{attribute addProperty BoxType "EK1100-0000-0018"}
{attribute addProperty Id "Beckhoff_EL73xxEK1122Beckhoff_EL73xxEK1122_FBF14708162A_0001_EL7332_0000_0016EL7332_BC9603EB19424.25A_0002_EL7332_0000_0017EL7332_BC9603EB19424.25A_0003_EL7332_0000_0018EL7332_BC9603EB19424.25A_0004_EL7332_0000_0019EL7332_BC9603EB19424.25A_0005_EL7332_0000_0020EL7332_BC9603EB19424.25A_0006_EL7332_0000_0021EL7332_BC9603EB19424.25A_0007_EL7332_0000_0022EL7332_BC9603EB19424.25A_0008_EL7332_0000_0023EL7332_20B9391519424.25A_0009_EL7332_0000_0024EL7332_20B9391519424.25A_0010_EL7342_0000_0016EL7342_E03DC37137046.25A_0011_EL7342_0000_0017EL7342_E03DC37137046.25A_0012_EL7342_0000_0018EL7342_E03DC37137046.25A_0013_EL7342_0000_0019EL7342_E03DC37137046.25A_0014_EL7342_0000_0020EL7342_E2585B8337046.25A_0015_EL7342_0000_0021EL7342_E2585B8337046.25A_0016_EL7342_0000_0022EL7342_E2585B8337046.25A_0017_EL7342_0000_0023EL7342_D8FCBEED37046.25A_0018_EL7342_0035_0019EL7342_E03DC37137046.25A_0019_EL7342_0035_0020EL7342_E03DC37137046.25"}
{attribute addProperty CRC "2633030660"}
{attribute addProperty SizeInBites "5462"}
{attribute addProperty SizeInBytes "682.75"}
TYPE Beckhoff_EL73xx_9CF0DC04 EXTENDS EK1100_179A0949 :
STRUCT
	{attribute addProperty Name "Beckhoff_EL73xxEK1122"}
	Beckhoff_EL73xxEK1122 : Beckhoff_EL73xxEK1122_FBF14708;
	{attribute addProperty Name "A_0001_EL7332_0000_0016"}
	A_0001_EL7332_0000_0016 : EL7332_BC9603EB;
	{attribute addProperty Name "A_0002_EL7332_0000_0017"}
	A_0002_EL7332_0000_0017 : EL7332_BC9603EB;
	{attribute addProperty Name "A_0003_EL7332_0000_0018"}
	A_0003_EL7332_0000_0018 : EL7332_BC9603EB;
	{attribute addProperty Name "A_0004_EL7332_0000_0019"}
	A_0004_EL7332_0000_0019 : EL7332_BC9603EB;
	{attribute addProperty Name "A_0005_EL7332_0000_0020"}
	A_0005_EL7332_0000_0020 : EL7332_BC9603EB;
	{attribute addProperty Name "A_0006_EL7332_0000_0021"}
	A_0006_EL7332_0000_0021 : EL7332_BC9603EB;
	{attribute addProperty Name "A_0007_EL7332_0000_0022"}
	A_0007_EL7332_0000_0022 : EL7332_BC9603EB;
	{attribute addProperty Name "A_0008_EL7332_0000_0023"}
	A_0008_EL7332_0000_0023 : EL7332_20B93915;
	{attribute addProperty Name "A_0009_EL7332_0000_0024"}
	A_0009_EL7332_0000_0024 : EL7332_20B93915;
	{attribute addProperty Name "A_0010_EL7342_0000_0016"}
	A_0010_EL7342_0000_0016 : EL7342_E03DC371;
	{attribute addProperty Name "A_0011_EL7342_0000_0017"}
	A_0011_EL7342_0000_0017 : EL7342_E03DC371;
	{attribute addProperty Name "A_0012_EL7342_0000_0018"}
	A_0012_EL7342_0000_0018 : EL7342_E03DC371;
	{attribute addProperty Name "A_0013_EL7342_0000_0019"}
	A_0013_EL7342_0000_0019 : EL7342_E03DC371;
	{attribute addProperty Name "A_0014_EL7342_0000_0020"}
	A_0014_EL7342_0000_0020 : EL7342_E2585B83;
	{attribute addProperty Name "A_0015_EL7342_0000_0021"}
	A_0015_EL7342_0000_0021 : EL7342_E2585B83;
	{attribute addProperty Name "A_0016_EL7342_0000_0022"}
	A_0016_EL7342_0000_0022 : EL7342_E2585B83;
	{attribute addProperty Name "A_0017_EL7342_0000_0023"}
	A_0017_EL7342_0000_0023 : EL7342_D8FCBEED;
	{attribute addProperty Name "A_0018_EL7342_0035_0019"}
	A_0018_EL7342_0035_0019 : EL7342_E03DC371;
	{attribute addProperty Name "A_0019_EL7342_0035_0020"}
	A_0019_EL7342_0035_0020 : EL7342_E03DC371;
END_STRUCT
END_TYPE

(* stored: Version 1.2.0.0, ProductVersion 3.1.4024.9
   DUT Beckhoff_EL73xx_9CF0DC04: Id {a5ad874d-e9f1-4005-beec-4e9307f466de} *)
